// TIA Portal project "Lab4" (V15.1)

(* hardware
DEVICE "S7-1200 station_2"  S7-1200 Station
   slot 0: "Rack_0"  S7-1200 Rack  Rack  V1.0
   slot 1: "PLC_1"  CPU 1214C AC/DC/Rly  6ES7 214-1BG31-0XB0  V3.0
   slot 3: "AQ 1x12BIT_1"  AQ1 signal board  6ES7 232-4HA30-0XB0  V1.0
*)

// ===== PLC "PLC_1"  CPU 1214C AC/DC/Rly =====

VAR_GLOBAL   // PLC tag table "Default tag table"
   "X_Level_Tank1" AT %IW64 : Int;   // Calle was here
   "Y_Level_Tank1" AT %QW80 : Int;
   "S1" AT %I0.0 : Bool;   // Sudden setpoing chane filling level 0 (0) or 700
END_VAR

ORGANIZATION_BLOCK "Main"   // OB1, LAD, ProgramCycle
TITLE = "Main Program Sweep (Cycle)"
{ S7_Optimized_Access := 'TRUE' }
VERSION : 0.1
BEGIN
END_ORGANIZATION_BLOCK

ORGANIZATION_BLOCK "Cyclic interrupt"   // OB30, LAD, CyclicInterrupt
TITLE = tank level control
{ S7_Optimized_Access := 'TRUE' }
VERSION : 0.1
   VAR_INPUT
      Initial_Call : Bool;   // Initial call of this OB
      Event_Count : Int;   // Events discarded
   END_VAR
   VAR_TEMP
      w_level_tank1 : Real;   // setpoint filling level tank1
   END_VAR
BEGIN

REGION Network 1: setpoint filling level 0 liter
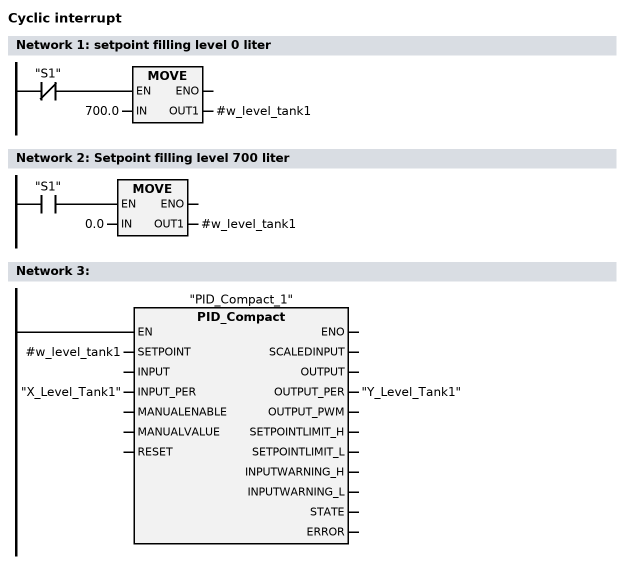
   RUNG wire#powerrail
      I_Contact( "S1" )
      { S7_GenerateENO := "TRUE" } Move(in := 700.0, out1 => #w_level_tank1)
   END_RUNG
   // the same network as SCL:
   IF NOT "S1" THEN #w_level_tank1 := 700.0; END_IF;
END_REGION

REGION Network 2: Setpoint filling level 700 liter
   RUNG wire#powerrail
      Contact( "S1" )
      { S7_GenerateENO := "TRUE" } Move(in := 0.0, out1 => #w_level_tank1)
   END_RUNG
   // the same network as SCL:
   IF "S1" THEN #w_level_tank1 := 0.0; END_IF;
END_REGION

REGION Network 3
   "PID_Compact_1"(Setpoint := #w_level_tank1, Input_PER := "X_Level_Tank1", Output_PER => "Y_Level_Tank1");   // PID_Compact
END_REGION
END_ORGANIZATION_BLOCK